ABB RobotStudio station: setupexample.rsstn

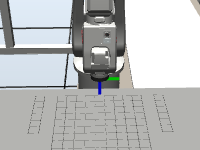
Station Station (saved by RobotStudio 6.7.7936.1011)
Controller MTRN4230, task T_ROB1: task frame (RAPID world) sits at (2935, -1760, 590) mm in the station
Controller MTRN4230
  mechanical unit ROB_1: IRB120_3_58__01, 6 joints, base frame (0, 0, 0) mm
Layout (positions relative to the parent item):
  - IRB120_3_58__01 [mechanism, from Robots\IRB120_3_58_G_01.rslib] at (2935, -1760, 590) mm; joint values [0, 0.1132, 1.2005, 0, 0.2571, 0] (rad or m)
  - ROBOTROOM [part] at (3020, -2855, 1950) mm, rotated rx 90 ry 0 rz 0 deg
  - Frame_1 [frame] at (0, 2854.49, -1444.72) mm, rotated rx 90 ry 0 rz 0 deg
